{attribute 'qualified_only'}
{attribute 'strict'}
TYPE e_MCState :
(
	Busy,
	Done,
	Error,
	CommandAborted,
	Active,
	Idle
);
END_TYPE

(* stored: Version 1.1.0.1, ProductVersion 3.1.4024.12
   DUT e_MCState: Id {dccfd427-6f0a-48c0-b6ce-5e9377677f3b} *)
